FUNCTION alg_a_Hstartled : BOOL
VAR_INPUT
	state: STATE;
END_VAR

alg_a_Hstartled := FALSE;

END_FUNCTION

(* stored: Version 1.1.0.1, ProductVersion 3.1.4022.18
   POU alg_a_Hstartled: Id {57467012-36d3-4110-aef0-5c334602d6ba}, SpecialFunc None *)
